TYPE HARDWAREGRP : UINT; END_TYPE

(* stored: Version 1.1.0.1, ProductVersion 3.1.0.25
   DUT HARDWAREGRP: Id {60fe8c73-27ac-437c-a638-4b02e2e8623b} *)
